// TIA Portal V20 export
DATA_BLOCK "TestVarIdent"   // DB76
TITLE = Test tags for ident
AUTHOR : SICAR
FAMILY : Ident
VERSION : 1.0
// Test tags for ident
// stored: MemoryReserve 100
   VAR
      init1 : Bool;   // Init 1
      read1 : Bool;   // Read1
      write1 : Bool;   // Write1
      init2 : Bool;   // Init 2
      read2 : Bool;   // Read2
      write2 : Bool;   // Write2
      testString : String[32];   // Test string
      charArr : Array[1..32] of Byte;   // Character Array
      prgNoMan : USInt;   // Program number manual
      enableManCtrlRf : Bool := false;   // Enable manual control RFID
      enableOption : Bool;   // Enable options
      enableManCtrlMV : Bool;   // Enable manual control MV
   END_VAR
BEGIN
END_DATA_BLOCK
